TYPE st_ManualDigitalMotorControl : // commands from manual controller
STRUCT
	bManRunCW 		: BOOL ;
	bManRunCWFast	: BOOL ;
	bManRunCCw		: BOOL ;
	bManRunCCWFast	: BOOL ; 
END_STRUCT
END_TYPE

(* stored: Version 1.1.0.1, ProductVersion 3.1.4024.10
   DUT st_ManualDigitalMotorControl: Id {162f917f-988a-0d87-1e32-0b4813687637} *)
